// Mitsubishi GX Works2 project: Cutter   PLC: FX1N/FX1NC

// global labels: Global1
VAR_GLOBAL
  FeedSpeedX AT D10 : DINT;
  CurrentX AT D2 : DINT;
  CurrentY AT D6 : DINT;
  FeedSpeedY AT D12 : DINT;
  OOnOffX AT Y024 : BOOL;
  OOnOffY AT Y026 : BOOL;
  OResetX AT Y025 : BOOL;
  OResetY AT Y027 : BOOL;
  ILimitReachedNX AT X010 : BOOL;
  ILimitReachedPX AT X011 : BOOL;
  ILimitReachedNY AT X030 : BOOL;
  ILimitReachedPY AT X031 : BOOL;
  PulseOutAndLimitX : PulseOutAndLimit;
  PulseOutAndLimitY : PulseOutAndLimit;
  OriginSetMove : OriginSetMove;
  RunButton AT M8 : BOOL;
  ManualYP AT M1 : BOOL;
  ManualYN AT M6 : BOOL;
  IsOn AT M0 : BOOL;
  LimitReachedX : BOOL;
  LimitReachedY : BOOL;
  TargetY AT D8 : DINT;
  ResetButton AT M2 : BOOL;
  OPulseX AT Y000 : BOOL;
  OPulseY AT Y001 : BOOL;
  ODirectionX AT Y002 : BOOL;
  ODirectionY AT Y003 : BOOL;
  StopButton AT M9 : BOOL;
  SetButton AT M5 : BOOL;
  OriginButton AT M7 : BOOL;
  TargetX AT D4 : DINT;
  ManualHandler : ManualHandler;
  OnOffResetStop : OnOffResetStop;
  ManualXP AT M4 : BOOL;
  ManualXN AT M3 : BOOL;
  DirectionX : BOOL;
  DirectionY : BOOL;
  CurrentPulseX AT D8140 : DINT;
  CurrentPulseY AT D8142 : DINT;
  DeltaX : DINT;
  DeltaY : DINT;
  MinX : DINT;
  MinY : DINT;
  MaxX : DINT;
  MaxY : DINT;
  FeedSpeed AT D0 : DINT;
  TargetReachedX : BOOL;
  TargetReachedY : BOOL;
  TargetReached : BOOL;
  AutoHandler : AutoHandler;
  PositionUpdater : PositionUpdater;
  RunButtonRisingLatch : BOOL;
  ManualX : BOOL;
  ManualY : BOOL;
  CommandId : INT;
  CommandNb : INT;
  OLazer AT Y004 : BOOL;
  AcDcTimeX AT D14 : DINT;
  AcDcTimeY AT D16 : DINT;
  RunButtonFallingLatch : BOOL;
  ArrayEnded AT M11 : BOOL;
  CommandIdArray AT D20 : ARRAY [0..49] OF INT;
  CommandNbArray AT D70 : ARRAY [0..49] OF INT;
  TargetArrayX AT D120 : ARRAY [0..49] OF DINT;
  TargetArrayY AT D220 : ARRAY [0..49] OF DINT;
  FeedSpeedArrayX AT D320 : ARRAY [0..49] OF DINT;
  FeedSpeedArrayY AT D420 : ARRAY [0..49] OF DINT;
  RunLatchX : BOOL;
  RunLatchY : BOOL;
  AutoNextLine AT M10 : BOOL;
END_VAR

// task Task_01 (event TRUE, interval 0, priority 31): POU_01

PROGRAM POU_01
VAR
  fTargetReachedRising : BOOL;
END_VAR
OnOffResetStop();

IF IsOn THEN
	PositionUpdater();
	ManualHandler();
	AutoHandler();

	PulseOutAndLimitX(
		fRunStart:= RunButtonRisingLatch, fManual:= ManualX, fTargetReached:= TargetReachedX, fRunLatch:= RunLatchX,
		fDirection:= DirectionX, fLimitReachedP:= NOT ILimitReachedPX, fLimitReachedN:= NOT ILimitReachedNX,
		fPulseFrequency:= FeedSpeedX, fPulseCount:= ABS(DeltaX), fAcDcTime:= AcDcTimeX,
		fOPulse:= OPulseX, fODirection:= ODirectionX);
	PulseOutAndLimitY(
		fRunStart:= RunButtonRisingLatch, fManual:= ManualY, fTargetReached:= TargetReachedY, fRunLatch:= RunLatchY,
		fDirection:= DirectionY, fLimitReachedP:= NOT ILimitReachedPY, fLimitReachedN:= NOT ILimitReachedNY,
		fPulseFrequency:= FeedSpeedY, fPulseCount:= ABS(DeltaY), fAcDcTime:= AcDcTimeY,
		fOPulse:= OPulseY, fODirection:= ODirectionY);
	
	RunButtonRisingLatch := FALSE;
	RunButtonFallingLatch := FALSE;
	SET(TargetReachedX AND TargetReachedY, TargetReached);
	PLS(TargetReached, fTargetReachedRising);
	RST(fTargetReachedRising, RunButton);
	
	OriginSetMove();
END_IF;
END_PROGRAM

FUNCTION_BLOCK PulseOutAndLimit
VAR_INPUT
  fLimitReachedP : BOOL;
  fLimitReachedN : BOOL;
  fPulseFrequency : DINT;
END_VAR
VAR
  fLimitReached : BOOL;
END_VAR
VAR_INPUT
  fDirection : BOOL;
  fAcDcTime : DINT;
END_VAR
VAR_OUTPUT
  fODirection : BOOL;
  fOPulse : BOOL;
END_VAR
VAR_INPUT
  fPulseCount : DINT;
  fManual : BOOL;
END_VAR
VAR_OUTPUT
  fTargetReached : BOOL;
END_VAR
VAR_INPUT
  fRunStart : BOOL;
END_VAR
VAR_IN_OUT
  fRunLatch : BOOL;
END_VAR
VAR
  fRunLatchFalling : BOOL;
END_VAR
RST(NOT fLimitReachedN AND NOT fLimitReachedP, fLimitReached);
RST(fLimitReachedN AND fDirection, fLimitReached);
RST(fLimitReachedP AND NOT fDirection, fLimitReached);

OUT(NOT fDirection, fODirection);
DPLSY(fManual AND NOT fLimitReached, fPulseFrequency, 0, fOPulse);

SET(fRunStart AND fPulseCount <> 0, fRunLatch);
DPLSR(fRunLatch, fPulseFrequency, fPulseCount, fAcDcTime, fOPulse);
RST(M8029, fRunLatch);
PLF(fRunLatch, fRunLatchFalling);
SET(fRunLatchFalling, fTargetReached);

SET(fLimitReachedN AND NOT fDirection, fLimitReached);
SET(fLimitReachedP AND fDirection, fLimitReached);
END_FUNCTION_BLOCK

FUNCTION_BLOCK OnOffResetStop
OUT(IsOn, OOnOffX);
OUT(IsOn, OOnOffY);

SET(ResetButton, OResetX);
SET(ResetButton, OResetY);
OUT_T(ResetButton, TC200, 8);
RST(TC200, ResetButton);
RST(TC200, OResetX);
RST(TC200, OResetY);

RST(StopButton, RunButton);
RST(StopButton, AutoNextLine);
RST(StopButton, RunLatchX);
RST(StopButton, RunLatchY);
RST(StopButton, StopButton);
END_FUNCTION_BLOCK

FUNCTION_BLOCK OriginSetMove
VAR
  SetOrigin : BOOL;
  MoveToOrigin : BOOL;
END_VAR
OUT(OriginButton AND SetButton, SetOrigin);
OUT(OriginButton AND NOT SetButton, MoveToOrigin);

RST(SetOrigin, CurrentX);
RST(SetOrigin, CurrentY);
RST(SetOrigin, CurrentPulseX);
RST(SetOrigin, CurrentPulseY);
RST(SetOrigin, SetButton);

RST(MoveToOrigin, TargetX);
RST(MoveToOrigin, TargetY);
SET(MoveToOrigin, RunButton);

RST(SetOrigin OR MoveToOrigin, OriginButton);
END_FUNCTION_BLOCK

FUNCTION_BLOCK ManualHandler
IF NOT RunButton THEN
	SET(ManualXP, DirectionX);
	RST(ManualXN, DirectionX);
	SET(ManualYP, DirectionY);
	RST(ManualYN, DirectionY);
	ManualX := ManualXP OR ManualXN;
	ManualY := ManualYP OR ManualYN;
	FeedSpeedX := FeedSpeed;
	FeedSpeedY := FeedSpeed;
ELSE
	ManualX := FALSE;
	ManualY := FALSE;
END_IF;
END_FUNCTION_BLOCK

FUNCTION_BLOCK AutoHandler
VAR
  fRBRising : BOOL;
  fRBFalling : BOOL;
  fIndex : INT;
END_VAR
PLS(RunButton, fRBRising);
SET(fRBRising, RunButtonRisingLatch);
PLF(RunButton, fRBFalling);
SET(fRBFalling, RunButtonFallingLatch);

IF RunButtonRisingLatch THEN
	SET(CommandId = 77 AND CommandNb = 3, OLazer);
	RST(CommandId = 77 AND CommandNb = 5, OLazer);
	
	DeltaX := TargetX - CurrentX;
	DeltaY := TargetY - CurrentY;
	DirectionX := DeltaX > 0;
	DirectionY := DeltaY > 0;
	TargetReachedX := DeltaX = 0;
	TargetReachedY := DeltaY = 0;
	
	TargetReached := TargetReachedX AND TargetReachedY;
	RST(TargetReached, RunButton);
END_IF;

IF RunButtonFallingLatch AND AutoNextLine THEN
	SET(fIndex > 3, ArrayEnded);
	RST(ArrayEnded, fIndex);
	CommandId := CommandIdArray[fIndex];
	CommandNb := CommandNbArray[fIndex];
	TargetX := TargetArrayX[fIndex];
	TargetY := TargetArrayY[fIndex];
	FeedSpeedX := FeedSpeedArrayX[fIndex];
	FeedSpeedY := FeedSpeedArrayY[fIndex];
	INC(NOT ArrayEnded, fIndex);
	SET(NOT ArrayEnded, RunButton);
END_IF;
END_FUNCTION_BLOCK

FUNCTION_BLOCK PositionUpdater
DADD(DirectionX, CurrentX, CurrentPulseX, CurrentX);
DSUB(NOT DirectionX, CurrentX, CurrentPulseX, CurrentX);
RST(TRUE, CurrentPulseX);
DADD(DirectionY, CurrentY, CurrentPulseY, CurrentY);
DSUB(NOT DirectionY, CurrentY, CurrentPulseY, CurrentY);
RST(TRUE, CurrentPulseY);
END_FUNCTION_BLOCK
